TYPE ST_ComauControl :
STRUCT
	q: ARRAY[0..2] OF LREAL;
	q_t: ARRAY[0..2] OF LREAL;
	q_tt: ARRAY[0..2] OF LREAL;
END_STRUCT
END_TYPE

(* stored: Version 1.1.0.1, ProductVersion 3.1.4022.7
   DUT ST_ComauControl: Id {141edc7e-e7a2-4a63-8f41-2c0c6574dcf6} *)
